FUNCTION_BLOCK T_TestEventHandler IMPLEMENTS I_TestEventHandler
VAR
    _EventWasRaised : BOOL;
    _EventData : UDINT;
END_VAR

PROPERTY EventWasRaised : BOOL
GET
EventWasRaised := _EventWasRaised;
END_GET
END_PROPERTY

METHOD OnCustomEvent
VAR_INPUT
    EventArgs : I_StreamReader;
END_VAR
_EventData := EventArgs.Read_UDINT();
_EventWasRaised := TRUE;
END_METHOD

END_FUNCTION_BLOCK

(* stored: Version 1.1.0.1, ProductVersion 3.1.4024.4
   POU T_TestEventHandler: Id {36315b4e-37c1-4c38-88f5-c97569f2b457}, SpecialFunc None
   Property EventWasRaised: Id {1a063ee9-2120-4506-8a93-8dcfddd034b8}
   Get Get: Id {cad574e2-1332-40f8-a7ef-a515438a13c2}
   Method OnCustomEvent: Id {64ee71a2-9a17-4869-8f6f-33f3ec8ccbf6} *)
